ABB RAPID module: Laboratorio1

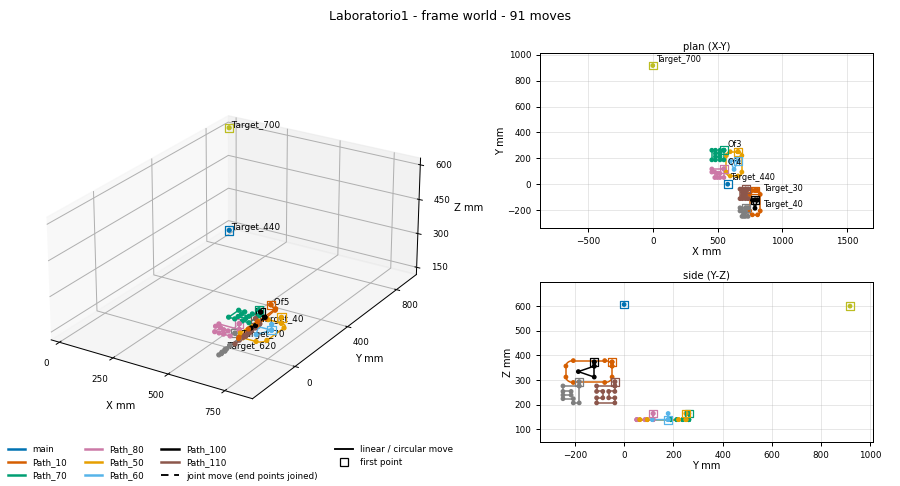
[picture p0: tool path of Laboratorio1 in frame world, 91 of 91 moves have a stored position in this frame; points joined in program order, loops and branches not executed]
MODULE Module1
        CONST robtarget Target_10:=[[48.75,212.044,0],[0,-0.707106781,0.707106781,0],[-1,-1,0,1],[9E+09,9E+09,9E+09,9E+09,9E+09,9E+09]];
    CONST robtarget Target_20:=[[57.537,233.258,0],[0,-0.707106781,0.707106781,0],[-1,-1,0,1],[9E+09,9E+09,9E+09,9E+09,9E+09,9E+09]];
    CONST robtarget Target_30:=[[78.75,242.044,0],[0,-0.707106781,0.707106781,0],[-1,-1,0,1],[9E+09,9E+09,9E+09,9E+09,9E+09,9E+09]];
    CONST robtarget Target_40:=[[206.25,242.044,0],[0,-0.707106781,0.707106781,0],[-1,-1,0,1],[9E+09,9E+09,9E+09,9E+09,9E+09,9E+09]];
    CONST robtarget Target_50:=[[227.463,233.258,0],[0,-0.707106781,0.707106781,0],[-1,-1,0,1],[9E+09,9E+09,9E+09,9E+09,9E+09,9E+09]];
    CONST robtarget Target_60:=[[236.25,212.044,0],[0,-0.707106781,0.707106781,0],[-1,-1,0,1],[9E+09,9E+09,9E+09,9E+09,9E+09,9E+09]];
    CONST robtarget Target_70:=[[236.25,152.044,0],[0,-0.707106781,0.707106781,0],[-1,-1,0,1],[9E+09,9E+09,9E+09,9E+09,9E+09,9E+09]];
    CONST robtarget Target_80:=[[227.463,130.831,0],[0,-0.707106781,0.707106781,0],[-1,-1,0,1],[9E+09,9E+09,9E+09,9E+09,9E+09,9E+09]];
    CONST robtarget Target_90:=[[206.25,122.044,0],[0,-0.707106781,0.707106781,0],[-1,-1,0,1],[9E+09,9E+09,9E+09,9E+09,9E+09,9E+09]];
    CONST robtarget Target_100:=[[78.75,122.044,0],[0,-0.707106781,0.707106781,0],[-1,-1,0,1],[9E+09,9E+09,9E+09,9E+09,9E+09,9E+09]];
    CONST robtarget Target_110:=[[57.537,130.831,0],[0,-0.707106781,0.707106781,0],[-1,-1,0,1],[9E+09,9E+09,9E+09,9E+09,9E+09,9E+09]];
    CONST robtarget Target_120:=[[48.75,152.044,0],[0,-0.707106781,0.707106781,0],[-1,-1,0,1],[9E+09,9E+09,9E+09,9E+09,9E+09,9E+09]];
    CONST robtarget Target_160:=[[121.29,211.777,0],[0,-0.707106781,0.707106781,0],[0,0,0,0],[9E+09,9E+09,9E+09,9E+09,9E+09,9E+09]];
    CONST robtarget Target_170:=[[185.79,181.777,0],[0,-0.707106781,0.707106781,0],[-1,0,1,0],[9E+09,9E+09,9E+09,9E+09,9E+09,9E+09]];
    CONST robtarget Target_180:=[[121.29,151.777,0],[0,-0.707106781,0.707106781,0],[-1,0,1,0],[9E+09,9E+09,9E+09,9E+09,9E+09,9E+09]];
    CONST robtarget Target_190:=[[37.639,103,0],[0,-0.707106781,0.707106781,0],[0,0,0,0],[9E+09,9E+09,9E+09,9E+09,9E+09,9E+09]];
    CONST robtarget Target_200:=[[111.639,103,0],[0,-0.707106781,0.707106781,0],[-1,0,1,0],[9E+09,9E+09,9E+09,9E+09,9E+09,9E+09]];
    CONST robtarget Target_210:=[[111.639,73,0],[0,-0.707106781,0.707106781,0],[-1,0,1,0],[9E+09,9E+09,9E+09,9E+09,9E+09,9E+09]];
    CONST robtarget Target_220:=[[86.639,73,0],[0,-0.707106781,0.707106781,0],[-1,0,1,0],[9E+09,9E+09,9E+09,9E+09,9E+09,9E+09]];
    CONST robtarget Target_230:=[[86.639,38,0],[0,-0.707106781,0.707106781,0],[-1,0,1,0],[9E+09,9E+09,9E+09,9E+09,9E+09,9E+09]];
    CONST robtarget Target_240:=[[111.639,38,0],[0,-0.707106781,0.707106781,0],[-1,0,1,0],[9E+09,9E+09,9E+09,9E+09,9E+09,9E+09]];
    CONST robtarget Target_250:=[[111.639,10,0],[0,-0.707106781,0.707106781,0],[-1,0,1,0],[9E+09,9E+09,9E+09,9E+09,9E+09,9E+09]];
    CONST robtarget Target_260:=[[37.639,10,0],[0,-0.707106781,0.707106781,0],[-1,0,1,0],[9E+09,9E+09,9E+09,9E+09,9E+09,9E+09]];
    CONST robtarget Target_270:=[[37.639,38,0],[0,-0.707106781,0.707106781,0],[-1,0,1,0],[9E+09,9E+09,9E+09,9E+09,9E+09,9E+09]];
    CONST robtarget Target_280:=[[62.639,38,0],[0,-0.707106781,0.707106781,0],[-1,0,1,0],[9E+09,9E+09,9E+09,9E+09,9E+09,9E+09]];
    CONST robtarget Target_290:=[[62.639,73,0],[0,-0.707106781,0.707106781,0],[-1,0,1,0],[9E+09,9E+09,9E+09,9E+09,9E+09,9E+09]];
    CONST robtarget Target_300:=[[37.639,73,0],[0,-0.707106781,0.707106781,0],[-1,0,1,0],[9E+09,9E+09,9E+09,9E+09,9E+09,9E+09]];
    CONST robtarget Target_310:=[[182.25,103,0],[0,-0.707106781,0.707106781,0],[0,0,0,0],[9E+09,9E+09,9E+09,9E+09,9E+09,9E+09]];
    CONST robtarget Target_320:=[[248.25,103,0],[0,-0.707106781,0.707106781,0],[-1,0,1,0],[9E+09,9E+09,9E+09,9E+09,9E+09,9E+09]];
    CONST robtarget Target_330:=[[248.25,73,0],[0,-0.707106781,0.707106781,0],[-1,0,1,0],[9E+09,9E+09,9E+09,9E+09,9E+09,9E+09]];
    CONST robtarget Target_340:=[[215.25,73,0],[0,-0.707106781,0.707106781,0],[-1,0,1,0],[9E+09,9E+09,9E+09,9E+09,9E+09,9E+09]];
    CONST robtarget Target_350:=[[215.25,53,0],[0,-0.707106781,0.707106781,0],[-1,0,1,0],[9E+09,9E+09,9E+09,9E+09,9E+09,9E+09]];
    CONST robtarget Target_360:=[[248.25,53,0],[0,-0.707106781,0.707106781,0],[0,0,0,0],[9E+09,9E+09,9E+09,9E+09,9E+09,9E+09]];
    CONST robtarget Target_370:=[[248.25,33,0],[0,-0.707106781,0.707106781,0],[0,0,0,0],[9E+09,9E+09,9E+09,9E+09,9E+09,9E+09]];
    CONST robtarget Target_380:=[[206.25,33,0],[0,-0.707106781,0.707106781,0],[0,0,0,0],[9E+09,9E+09,9E+09,9E+09,9E+09,9E+09]];
    CONST robtarget Target_390:=[[206.25,10,0],[0,-0.707106781,0.707106781,0],[0,0,0,0],[9E+09,9E+09,9E+09,9E+09,9E+09,9E+09]];
    CONST robtarget Target_400:=[[182.25,10,0],[0,-0.707106781,0.707106781,0],[0,0,0,0],[9E+09,9E+09,9E+09,9E+09,9E+09,9E+09]];
    CONST robtarget Target_410:=[[-200,618.426700281,73.425017241],[0.199173924,0.678476048,-0.678476048,0.199173924],[0,0,0,0],[9E+09,9E+09,9E+09,9E+09,9E+09,9E+09]];
    CONST robtarget Target_420:=[[37.639,103,10],[0,-0.707106781,0.707106781,0],[-1,0,1,0],[9E+09,9E+09,9E+09,9E+09,9E+09,9E+09]];
    CONST robtarget Target_430:=[[-150,450.239208352,258.39249427],[0,-0.707106781,0.707106781,0],[0,0,0,0],[9E+09,9E+09,9E+09,9E+09,9E+09,9E+09]];
    CONST robtarget Target_10_2:=[[48.75,212.044,0],[0,-0.707106781,0.707106781,0],[0,0,0,0],[9E+09,9E+09,9E+09,9E+09,9E+09,9E+09]];
    CONST robtarget Target_20_2:=[[57.537,233.258,0],[0,-0.707106781,0.707106781,0],[0,-1,1,0],[9E+09,9E+09,9E+09,9E+09,9E+09,9E+09]];
    CONST robtarget Target_30_2:=[[78.75,242.044,0],[0,-0.707106781,0.707106781,0],[0,-1,1,0],[9E+09,9E+09,9E+09,9E+09,9E+09,9E+09]];
    CONST robtarget Target_40_2:=[[206.25,242.044,0],[0,-0.707106781,0.707106781,0],[0,-2,1,0],[9E+09,9E+09,9E+09,9E+09,9E+09,9E+09]];
    CONST robtarget Target_50_2:=[[227.463,233.258,0],[0,-0.707106781,0.707106781,0],[0,-2,1,0],[9E+09,9E+09,9E+09,9E+09,9E+09,9E+09]];
    CONST robtarget Target_60_2:=[[236.25,212.044,0],[0,-0.707106781,0.707106781,0],[0,-2,1,0],[9E+09,9E+09,9E+09,9E+09,9E+09,9E+09]];
    CONST robtarget Target_70_2:=[[236.25,152.044,0],[0,-0.707106781,0.707106781,0],[0,-2,1,0],[9E+09,9E+09,9E+09,9E+09,9E+09,9E+09]];
    CONST robtarget Target_80_2:=[[227.463,130.831,0],[0,-0.707106781,0.707106781,0],[0,-2,1,0],[9E+09,9E+09,9E+09,9E+09,9E+09,9E+09]];
    CONST robtarget Target_90_2:=[[206.25,122.044,0],[0,-0.707106781,0.707106781,0],[0,-2,1,0],[9E+09,9E+09,9E+09,9E+09,9E+09,9E+09]];
    CONST robtarget Target_100_2:=[[78.75,122.044,0],[0,-0.707106781,0.707106781,0],[0,-2,1,0],[9E+09,9E+09,9E+09,9E+09,9E+09,9E+09]];
    CONST robtarget Target_110_2:=[[57.537,130.831,0],[0,-0.707106781,0.707106781,0],[0,-2,1,0],[9E+09,9E+09,9E+09,9E+09,9E+09,9E+09]];
    CONST robtarget Target_120_2:=[[48.75,152.044,0],[0,-0.707106781,0.707106781,0],[0,-2,1,0],[9E+09,9E+09,9E+09,9E+09,9E+09,9E+09]];
    CONST robtarget Target_160_2:=[[121.29,211.777,0],[0,-0.707106781,0.707106781,0],[0,-2,1,0],[9E+09,9E+09,9E+09,9E+09,9E+09,9E+09]];
    CONST robtarget Target_170_2:=[[185.79,181.777,0],[0,-0.707106781,0.707106781,0],[0,-2,1,0],[9E+09,9E+09,9E+09,9E+09,9E+09,9E+09]];
    CONST robtarget Target_180_2:=[[121.29,151.777,0],[0,-0.707106781,0.707106781,0],[0,-2,1,0],[9E+09,9E+09,9E+09,9E+09,9E+09,9E+09]];
    CONST robtarget Target_190_2:=[[37.639,103,0],[0,-0.707106781,0.707106781,0],[0,-2,1,0],[9E+09,9E+09,9E+09,9E+09,9E+09,9E+09]];
    CONST robtarget Target_200_2:=[[111.639,103,0],[0,-0.707106781,0.707106781,0],[0,-2,1,0],[9E+09,9E+09,9E+09,9E+09,9E+09,9E+09]];
    CONST robtarget Target_210_2:=[[111.639,73,0],[0,-0.707106781,0.707106781,0],[0,-2,1,0],[9E+09,9E+09,9E+09,9E+09,9E+09,9E+09]];
    CONST robtarget Target_220_2:=[[86.639,73,0],[0,-0.707106781,0.707106781,0],[0,-2,1,0],[9E+09,9E+09,9E+09,9E+09,9E+09,9E+09]];
    CONST robtarget Target_230_2:=[[86.639,38,0],[0,-0.707106781,0.707106781,0],[0,-2,1,0],[9E+09,9E+09,9E+09,9E+09,9E+09,9E+09]];
    CONST robtarget Target_240_2:=[[111.639,38,0],[0,-0.707106781,0.707106781,0],[0,-2,1,0],[9E+09,9E+09,9E+09,9E+09,9E+09,9E+09]];
    CONST robtarget Target_250_2:=[[111.639,10,0],[0,-0.707106781,0.707106781,0],[0,-2,1,0],[9E+09,9E+09,9E+09,9E+09,9E+09,9E+09]];
    CONST robtarget Target_260_2:=[[37.639,10,0],[0,-0.707106781,0.707106781,0],[0,-2,1,0],[9E+09,9E+09,9E+09,9E+09,9E+09,9E+09]];
    CONST robtarget Target_270_2:=[[37.639,38,0],[0,-0.707106781,0.707106781,0],[0,-2,1,0],[9E+09,9E+09,9E+09,9E+09,9E+09,9E+09]];
    CONST robtarget Target_280_2:=[[62.639,38,0],[0,-0.707106781,0.707106781,0],[0,-2,1,0],[9E+09,9E+09,9E+09,9E+09,9E+09,9E+09]];
    CONST robtarget Target_290_2:=[[62.639,73,0],[0,-0.707106781,0.707106781,0],[0,-2,1,0],[9E+09,9E+09,9E+09,9E+09,9E+09,9E+09]];
    CONST robtarget Target_300_2:=[[37.639,73,0],[0,-0.707106781,0.707106781,0],[0,-2,1,0],[9E+09,9E+09,9E+09,9E+09,9E+09,9E+09]];
    CONST robtarget Target_310_2:=[[182.25,103,0],[0,-0.707106781,0.707106781,0],[0,-2,1,0],[9E+09,9E+09,9E+09,9E+09,9E+09,9E+09]];
    CONST robtarget Target_320_2:=[[248.25,103,0],[0,-0.707106781,0.707106781,0],[0,-2,1,0],[9E+09,9E+09,9E+09,9E+09,9E+09,9E+09]];
    CONST robtarget Target_330_2:=[[248.25,73,0],[0,-0.707106781,0.707106781,0],[0,-2,1,0],[9E+09,9E+09,9E+09,9E+09,9E+09,9E+09]];
    CONST robtarget Target_340_2:=[[215.25,73,0],[0,-0.707106781,0.707106781,0],[0,-2,1,0],[9E+09,9E+09,9E+09,9E+09,9E+09,9E+09]];
    CONST robtarget Target_350_2:=[[215.25,53,0],[0,-0.707106781,0.707106781,0],[0,-2,1,0],[9E+09,9E+09,9E+09,9E+09,9E+09,9E+09]];
    CONST robtarget Target_360_2:=[[248.25,53,0],[0,-0.707106781,0.707106781,0],[0,-2,1,0],[9E+09,9E+09,9E+09,9E+09,9E+09,9E+09]];
    CONST robtarget Target_370_2:=[[248.25,33,0],[0,-0.707106781,0.707106781,0],[0,-2,1,0],[9E+09,9E+09,9E+09,9E+09,9E+09,9E+09]];
    CONST robtarget Target_380_2:=[[206.25,33,0],[0,-0.707106781,0.707106781,0],[0,-2,1,0],[9E+09,9E+09,9E+09,9E+09,9E+09,9E+09]];
    CONST robtarget Target_390_2:=[[206.25,10,0],[0,-0.707106781,0.707106781,0],[0,-2,1,0],[9E+09,9E+09,9E+09,9E+09,9E+09,9E+09]];
    CONST robtarget Target_400_2:=[[182.25,10,0],[0,-0.707106781,0.707106781,0],[0,-2,1,0],[9E+09,9E+09,9E+09,9E+09,9E+09,9E+09]];
    CONST robtarget Target_440:=[[300,132.895467338,467.521656757],[0.092171548,-0.701073752,0.701073752,0.092171548],[0,0,0,0],[9E+09,9E+09,9E+09,9E+09,9E+09,9E+09]];
    CONST robtarget Target_450:=[[121.29,211.777,0],[0,-0.707106781,0.707106781,0],[-1,-1,0,1],[9E+09,9E+09,9E+09,9E+09,9E+09,9E+09]];
    PERS tooldata MyNewTool:=[TRUE,[[113.137,0,149.137],[0.923879533,0,0.382683432,0]],[1,[0,0,1],[1,0,0,0],0,0,0]];
    TASK PERS wobjdata Workobject_4:=[FALSE,TRUE,"",[[250,50,250],[1,0,0,0]],[[417.158,-50,-50],[0.646674178,0.286028859,-0.286028859,-0.646674178]]];
    TASK PERS wobjdata Workobject_4_2:=[FALSE,TRUE,"",[[300,500,300],[0.91460716,0,0.404343596,0]],[[217.158,-200,0],[0.646674178,0.286028859,-0.286028859,-0.646674178]]];
    CONST robtarget Target_460:=[[185.79,181.777,0],[0,-0.707106781,0.707106781,0],[-1,-1,0,1],[9E+09,9E+09,9E+09,9E+09,9E+09,9E+09]];
    CONST robtarget Target_420_2:=[[37.639,103,10],[0,-0.707106781,0.707106781,0],[0,-1,1,0],[9E+09,9E+09,9E+09,9E+09,9E+09,9E+09]];
    CONST robtarget Home:=[[-150,450.239208352,258.39249427],[0.199173924,0.678476048,-0.678476048,0.199173924],[0,0,0,0],[9E+09,9E+09,9E+09,9E+09,9E+09,9E+09]];
    CONST robtarget Target_470:=[[121.29,151.777,0],[0,-0.707106781,0.707106781,0],[-1,-1,0,1],[9E+09,9E+09,9E+09,9E+09,9E+09,9E+09]];
    CONST robtarget Target_480:=[[37.639,103,0],[0,-0.707106781,0.707106781,0],[-1,-1,0,1],[9E+09,9E+09,9E+09,9E+09,9E+09,9E+09]];
    CONST robtarget Target_490:=[[111.639,103,0],[0,-0.707106781,0.707106781,0],[-1,-1,0,1],[9E+09,9E+09,9E+09,9E+09,9E+09,9E+09]];
    CONST robtarget Target_500:=[[111.639,73,0],[0,-0.707106781,0.707106781,0],[-1,-1,0,1],[9E+09,9E+09,9E+09,9E+09,9E+09,9E+09]];
    CONST robtarget Target_510:=[[86.639,73,0],[0,-0.707106781,0.707106781,0],[-1,-1,0,1],[9E+09,9E+09,9E+09,9E+09,9E+09,9E+09]];
    CONST robtarget Target_520:=[[86.639,38,0],[0,-0.707106781,0.707106781,0],[-1,-1,0,1],[9E+09,9E+09,9E+09,9E+09,9E+09,9E+09]];
    CONST robtarget Target_530:=[[111.639,38,0],[0,-0.707106781,0.707106781,0],[-1,-1,0,1],[9E+09,9E+09,9E+09,9E+09,9E+09,9E+09]];
    CONST robtarget Target_540:=[[111.639,10,0],[0,-0.707106781,0.707106781,0],[-1,-1,0,1],[9E+09,9E+09,9E+09,9E+09,9E+09,9E+09]];
    CONST robtarget Target_550:=[[37.639,10,0],[0,-0.707106781,0.707106781,0],[-1,-1,0,1],[9E+09,9E+09,9E+09,9E+09,9E+09,9E+09]];
    CONST robtarget Target_560:=[[37.639,38,0],[0,-0.707106781,0.707106781,0],[-1,-1,0,1],[9E+09,9E+09,9E+09,9E+09,9E+09,9E+09]];
    CONST robtarget Target_570:=[[62.639,38,0],[0,-0.707106781,0.707106781,0],[-1,-1,0,1],[9E+09,9E+09,9E+09,9E+09,9E+09,9E+09]];
    CONST robtarget Target_580:=[[62.639,73,0],[0,-0.707106781,0.707106781,0],[-1,-1,0,1],[9E+09,9E+09,9E+09,9E+09,9E+09,9E+09]];
    CONST robtarget Target_590:=[[37.639,73,0],[0,-0.707106781,0.707106781,0],[-1,-1,0,1],[9E+09,9E+09,9E+09,9E+09,9E+09,9E+09]];
    CONST robtarget Target_600:=[[182.25,103,0],[0,-0.707106781,0.707106781,0],[-1,-1,0,1],[9E+09,9E+09,9E+09,9E+09,9E+09,9E+09]];
    CONST robtarget Target_610:=[[248.25,103,0],[0,-0.707106781,0.707106781,0],[-1,-1,0,1],[9E+09,9E+09,9E+09,9E+09,9E+09,9E+09]];
    CONST robtarget Target_620:=[[248.25,73,0],[0,-0.707106781,0.707106781,0],[-1,-1,0,1],[9E+09,9E+09,9E+09,9E+09,9E+09,9E+09]];
    CONST robtarget Target_630:=[[215.25,73,0],[0,-0.707106781,0.707106781,0],[-1,-1,0,1],[9E+09,9E+09,9E+09,9E+09,9E+09,9E+09]];
    CONST robtarget Target_640:=[[215.25,53,0],[0,-0.707106781,0.707106781,0],[-1,-1,0,1],[9E+09,9E+09,9E+09,9E+09,9E+09,9E+09]];
    CONST robtarget Target_650:=[[248.25,53,0],[0,-0.707106781,0.707106781,0],[-1,-1,0,1],[9E+09,9E+09,9E+09,9E+09,9E+09,9E+09]];
    CONST robtarget Target_660:=[[248.25,33,0],[0,-0.707106781,0.707106781,0],[-1,-1,0,1],[9E+09,9E+09,9E+09,9E+09,9E+09,9E+09]];
    CONST robtarget Target_670:=[[206.25,33,0],[0,-0.707106781,0.707106781,0],[-1,-1,0,1],[9E+09,9E+09,9E+09,9E+09,9E+09,9E+09]];
    CONST robtarget Target_680:=[[206.25,10,0],[0,-0.707106781,0.707106781,0],[-1,-1,0,1],[9E+09,9E+09,9E+09,9E+09,9E+09,9E+09]];
    CONST robtarget Target_690:=[[182.25,10,0],[0,-0.707106781,0.707106781,0],[-1,-1,0,1],[9E+09,9E+09,9E+09,9E+09,9E+09,9E+09]];
    CONST robtarget Target_700:=[[-916.996195421,-152.709286658,762.867669219],[0.373714714,0.844920531,-0.154797703,-0.349977543],[1,0,-1,0],[9E+09,9E+09,9E+09,9E+09,9E+09,9E+09]];
    CONST robtarget Of1:=[[48.75,212.044,25],[0,-0.707106781,0.707106781,0],[0,-1,0,0],[9E+09,9E+09,9E+09,9E+09,9E+09,9E+09]];
    CONST robtarget Of2:=[[121.29,211.777,25],[0,-0.707106781,0.707106781,0],[0,-1,0,0],[9E+09,9E+09,9E+09,9E+09,9E+09,9E+09]];
    CONST robtarget Of3:=[[37.639,103,25],[0,-0.707106781,0.707106781,0],[0,-1,1,0],[9E+09,9E+09,9E+09,9E+09,9E+09,9E+09]];
    CONST robtarget Of4:=[[182.25,103,25],[0,-0.707106781,0.707106781,0],[0,-2,1,0],[9E+09,9E+09,9E+09,9E+09,9E+09,9E+09]];
    CONST robtarget Of5:=[[48.75,212.044,25],[0,-0.707106781,0.707106781,0],[-1,-1,0,1],[9E+09,9E+09,9E+09,9E+09,9E+09,9E+09]];
    CONST robtarget Of6:=[[121.29,211.777,25],[0,-0.707106781,0.707106781,0],[-1,-1,0,1],[9E+09,9E+09,9E+09,9E+09,9E+09,9E+09]];
    CONST robtarget Of7:=[[37.639,103,25],[0,-0.707106781,0.707106781,0],[-1,-1,0,1],[9E+09,9E+09,9E+09,9E+09,9E+09,9E+09]];
    CONST robtarget Of8:=[[182.25,103,25],[0,-0.707106781,0.707106781,0],[-1,-1,0,1],[9E+09,9E+09,9E+09,9E+09,9E+09,9E+09]];
!***********************************************************
    !
    ! M?dulo:  Module1
    !
    ! Descripción:
    !   <Introduzca la descripción aquí>
    !
    ! Autor: ferna
    !
    ! Versión: 1.0
    !
    !***********************************************************


    !***********************************************************
    !
    ! Procedimiento Main
    !
    !   Este es el punto de entrada de su programa
    !
    !***********************************************************
    PROC main()
        SetDO DO_01,0;
        WHILE TRUE DO
            IF DI_01 = 1 THEN
                SetDO DO_01,1;
                Path_50;
                Path_60;
                Path_70;
                Path_80;
                Path_10;
                Path_100;
                Path_110;
                Path_120;
                MoveJ Target_440,v400,z0,MyNewTool\WObj:=Workobject_4_2;
            ENDIF
            IF DI_02 = 1 THEN
                SetDO DO_01,0;
                Path_130;
            ENDIF
        ENDWHILE
    ENDPROC
    PROC Path_10()
        MoveJ Of5,v400,z0,MyNewTool\WObj:=Workobject_4;
        MoveJ Target_10,v400,z0,MyNewTool\WObj:=Workobject_4;
        MoveC Target_20,Target_30,v100,z0,MyNewTool\WObj:=Workobject_4;
        MoveL Target_40,v100,z0,MyNewTool\WObj:=Workobject_4;
        MoveC Target_50,Target_60,v100,z0,MyNewTool\WObj:=Workobject_4;
        MoveL Target_70,v100,z0,MyNewTool\WObj:=Workobject_4;
        MoveC Target_80,Target_90,v100,z0,MyNewTool\WObj:=Workobject_4;
        MoveL Target_100,v100,z0,MyNewTool\WObj:=Workobject_4;
        MoveC Target_110,Target_120,v100,z0,MyNewTool\WObj:=Workobject_4;
        MoveL Target_10,v100,z0,MyNewTool\WObj:=Workobject_4;
        MoveJ Of5,v400,z0,MyNewTool\WObj:=Workobject_4;
    ENDPROC
    PROC Path_70()
        MoveJ Of3,v400,z0,MyNewTool\WObj:=Workobject_4_2;
        MoveJ Target_190_2,v400,z0,MyNewTool\WObj:=Workobject_4_2;
        MoveL Target_200_2,v100,z0,MyNewTool\WObj:=Workobject_4_2;
        MoveL Target_210_2,v100,z0,MyNewTool\WObj:=Workobject_4_2;
        MoveL Target_220_2,v100,z0,MyNewTool\WObj:=Workobject_4_2;
        MoveL Target_230_2,v100,z0,MyNewTool\WObj:=Workobject_4_2;
        MoveL Target_240_2,v100,z0,MyNewTool\WObj:=Workobject_4_2;
        MoveL Target_250_2,v100,z0,MyNewTool\WObj:=Workobject_4_2;
        MoveL Target_260_2,v100,z0,MyNewTool\WObj:=Workobject_4_2;
        MoveL Target_270_2,v100,z0,MyNewTool\WObj:=Workobject_4_2;
        MoveL Target_280_2,v100,z0,MyNewTool\WObj:=Workobject_4_2;
        MoveL Target_290_2,v100,z0,MyNewTool\WObj:=Workobject_4_2;
        MoveL Target_300_2,v100,z0,MyNewTool\WObj:=Workobject_4_2;
        MoveL Target_190_2,v100,z0,MyNewTool\WObj:=Workobject_4_2;
        MoveJ Of3,v400,z0,MyNewTool\WObj:=Workobject_4_2;
    ENDPROC
    PROC Path_80()
        MoveJ Of4,v400,z0,MyNewTool\WObj:=Workobject_4_2;
        MoveJ Target_310_2,v400,z0,MyNewTool\WObj:=Workobject_4_2;
        MoveL Target_320_2,v100,z0,MyNewTool\WObj:=Workobject_4_2;
        MoveL Target_330_2,v100,z0,MyNewTool\WObj:=Workobject_4_2;
        MoveL Target_340_2,v100,z0,MyNewTool\WObj:=Workobject_4_2;
        MoveL Target_350_2,v100,z0,MyNewTool\WObj:=Workobject_4_2;
        MoveL Target_360_2,v100,z0,MyNewTool\WObj:=Workobject_4_2;
        MoveL Target_370_2,v100,z0,MyNewTool\WObj:=Workobject_4_2;
        MoveL Target_380_2,v100,z0,MyNewTool\WObj:=Workobject_4_2;
        MoveL Target_390_2,v100,z0,MyNewTool\WObj:=Workobject_4_2;
        MoveL Target_400_2,v100,z0,MyNewTool\WObj:=Workobject_4_2;
        MoveL Target_310_2,v100,z0,MyNewTool\WObj:=Workobject_4_2;
        MoveJ Of4,v400,z0,MyNewTool\WObj:=Workobject_4_2;
    ENDPROC
    PROC Path_50()
        MoveJ Of1,v400,z0,MyNewTool\WObj:=Workobject_4_2;
        MoveJ Target_10_2,v400,z0,MyNewTool\WObj:=Workobject_4_2;
        MoveC Target_20_2,Target_30_2,v100,z0,MyNewTool\WObj:=Workobject_4_2;
        MoveL Target_40_2,v100,z0,MyNewTool\WObj:=Workobject_4_2;
        MoveC Target_50_2,Target_60_2,v100,z0,MyNewTool\WObj:=Workobject_4_2;
        MoveL Target_70_2,v100,z0,MyNewTool\WObj:=Workobject_4_2;
        MoveC Target_80_2,Target_90_2,v100,z0,MyNewTool\WObj:=Workobject_4_2;
        MoveL Target_100_2,v100,z0,MyNewTool\WObj:=Workobject_4_2;
        MoveC Target_110_2,Target_120_2,v100,z0,MyNewTool\WObj:=Workobject_4_2;
        MoveL Target_10_2,v100,z0,MyNewTool\WObj:=Workobject_4_2;
        MoveJ Of1,v400,z0,MyNewTool\WObj:=Workobject_4_2;
    ENDPROC
    PROC Path_60()
        MoveJ Target_160_2,v400,z0,MyNewTool\WObj:=Workobject_4_2;
        MoveL Target_170_2,v100,z0,MyNewTool\WObj:=Workobject_4_2;
        MoveL Target_180_2,v100,z0,MyNewTool\WObj:=Workobject_4_2;
        MoveL Target_160_2,v100,z0,MyNewTool\WObj:=Workobject_4_2;
        MoveJ Of2,v400,z0,MyNewTool\WObj:=Workobject_4_2;
    ENDPROC
    PROC Path_100()
        MoveJ Of6,v400,z0,MyNewTool\WObj:=Workobject_4;
        MoveJ Target_450,v400,z0,MyNewTool\WObj:=Workobject_4;
        MoveL Target_460,v100,z0,MyNewTool\WObj:=Workobject_4;
        MoveL Target_470,v100,z0,MyNewTool\WObj:=Workobject_4;
        MoveL Target_450,v100,z0,MyNewTool\WObj:=Workobject_4;
        MoveJ Of6,v400,z0,MyNewTool\WObj:=Workobject_4;
    ENDPROC
    PROC Path_110()
        MoveJ Of7,v400,z0,MyNewTool\WObj:=Workobject_4;
        MoveJ Target_480,v400,z0,MyNewTool\WObj:=Workobject_4;
        MoveL Target_490,v100,z0,MyNewTool\WObj:=Workobject_4;
        MoveL Target_500,v100,z0,MyNewTool\WObj:=Workobject_4;
        MoveL Target_510,v100,z0,MyNewTool\WObj:=Workobject_4;
        MoveL Target_520,v100,z0,MyNewTool\WObj:=Workobject_4;
        MoveL Target_530,v100,z0,MyNewTool\WObj:=Workobject_4;
        MoveL Target_540,v100,z0,MyNewTool\WObj:=Workobject_4;
        MoveL Target_550,v100,z0,MyNewTool\WObj:=Workobject_4;
        MoveL Target_560,v100,z0,MyNewTool\WObj:=Workobject_4;
        MoveL Target_570,v100,z0,MyNewTool\WObj:=Workobject_4;
        MoveL Target_580,v100,z0,MyNewTool\WObj:=Workobject_4;
        MoveL Target_590,v100,z0,MyNewTool\WObj:=Workobject_4;
        MoveL Target_480,v100,z0,MyNewTool\WObj:=Workobject_4;
        MoveJ Of7,v400,z0,MyNewTool\WObj:=Workobject_4;
    ENDPROC
    PROC Path_120()
        MoveJ Of8,v400,z0,MyNewTool\WObj:=Workobject_4;
        MoveJ Target_600,v400,z0,MyNewTool\WObj:=Workobject_4;
        MoveL Target_610,v100,z0,MyNewTool\WObj:=Workobject_4;
        MoveL Target_620,v100,z0,MyNewTool\WObj:=Workobject_4;
        MoveL Target_630,v100,z0,MyNewTool\WObj:=Workobject_4;
        MoveL Target_640,v100,z0,MyNewTool\WObj:=Workobject_4;
        MoveL Target_650,v100,z0,MyNewTool\WObj:=Workobject_4;
        MoveL Target_660,v100,z0,MyNewTool\WObj:=Workobject_4;
        MoveL Target_670,v100,z0,MyNewTool\WObj:=Workobject_4;
        MoveL Target_680,v100,z0,MyNewTool\WObj:=Workobject_4;
        MoveL Target_690,v100,z0,MyNewTool\WObj:=Workobject_4;
        MoveL Target_600,v100,z0,MyNewTool\WObj:=Workobject_4;
        MoveJ Of8,v400,z0,MyNewTool\WObj:=Workobject_4;
    ENDPROC
    PROC Path_130()
        MoveJ Target_700,v400,z0,MyNewTool\WObj:=Workobject_4;
    ENDPROC
ENDMODULE
